FUNCTION_BLOCK FB_System_BHKW_921
VAR
	Pumpe_321: FB_PU;
	Stellventil_321: FB_SVs;
	Regelventil_321: FB_RV;
	BHKW_921: FB_BHKW;
	Zustandscheck: FB_System_BHKW_Zustandscheck;
	Logik: FB_System_BHKW_Logik;
	Ablaufsteuerung: FB_System_BHKW_Ablaufsteuerung;
	Timer1: TON;
	Timer_BHKW921_Pumpe321_Freigabe: TOF;
	Sollwertscheck: FB_System_BHKW_Sollwertscheck;
END_VAR
VAR_INPUT
	Freigabe_auto: BOOL := TRUE;
	Betrieb_Anford_auto: BOOL := FALSE;
	Regelung_Sollw_auto: REAL := 60;
END_VAR
VAR_OUTPUT
	{attribute 'OPC.UA.DA' := '1'}Steuerung: ST_System_BHKW_Steuerung; 
	{attribute 'OPC.UA.DA' := '1'}Stellwert: ST_System_BHKW_Stellwert; 
	{attribute 'OPC.UA.DA' := '1'}Zustand: ST_System_BHKW_Zustand; 		
	{attribute 'OPC.UA.DA' := '1'}Parameter: ST_System_BHKW_Parameter; 
END_VAR
VAR // added by the converter: edge detectors and wires of the graphical bodies
    _w1, _w2, _w3, _w4 : ANY;
END_VAR

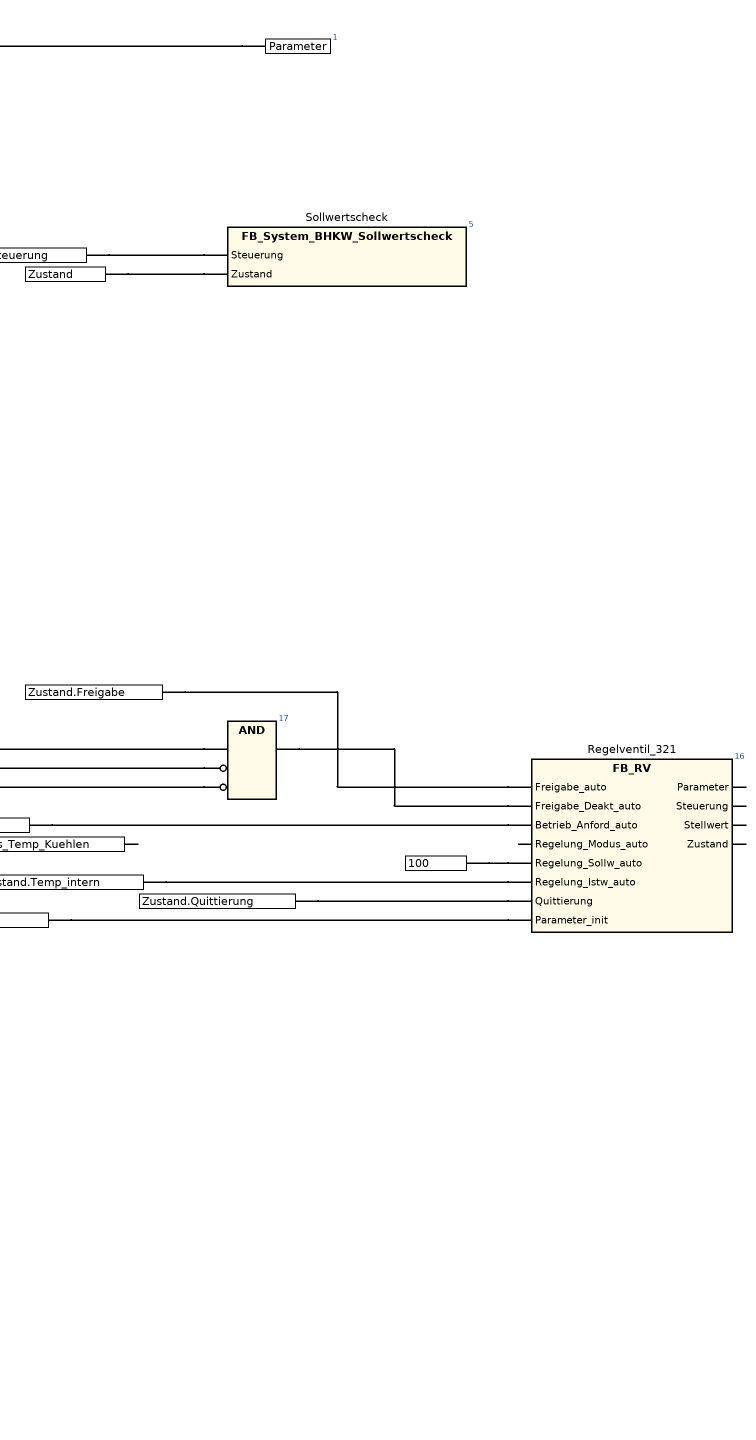
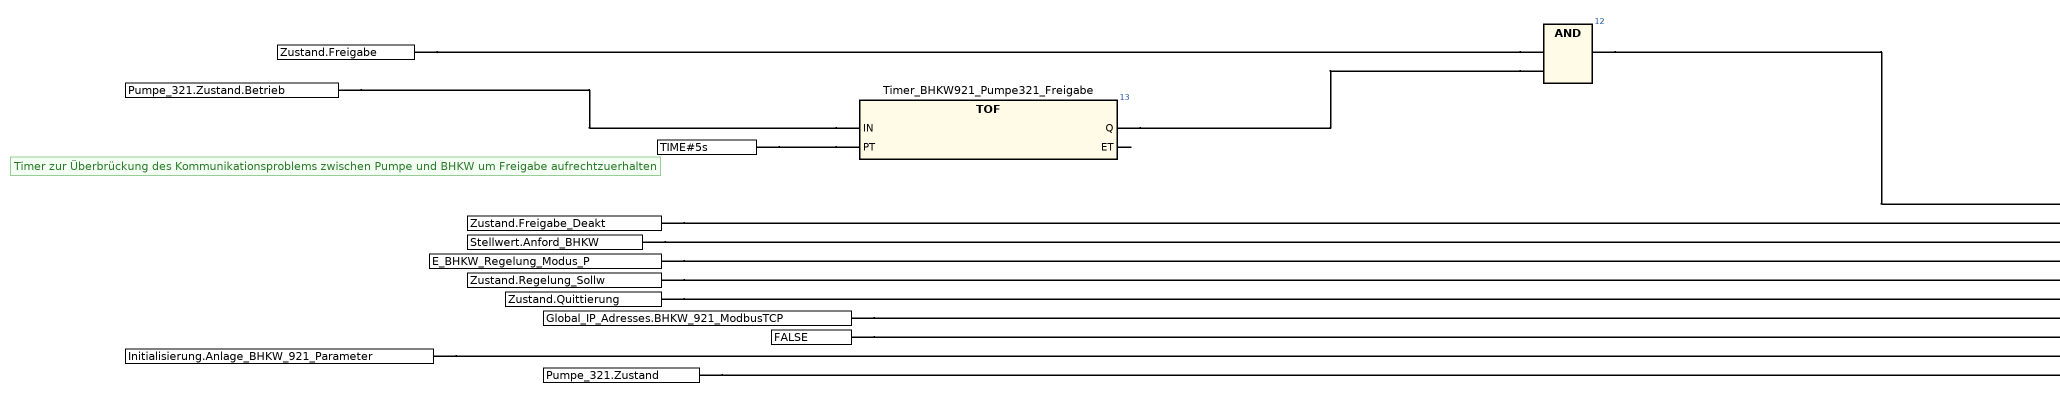
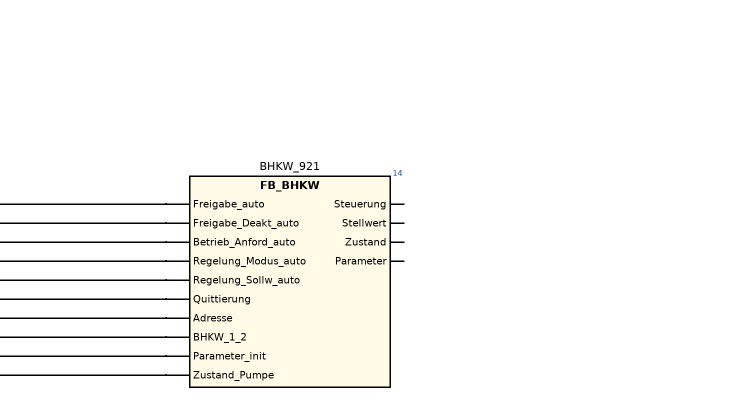
Steuerung.Freigabe.auto := Freigabe_auto;
Parameter := Initialisierung.System_BHKW_Parameter;
Steuerung.Freigabe_Deakt.auto := TRUE;
Steuerung.Betrieb_Anford.auto := Betrieb_Anford_auto;
Steuerung.Regelung_Sollw.auto := Regelung_Sollw_auto;
Sollwertscheck(Steuerung := Steuerung, Zustand := Zustand); // FB_System_BHKW_Sollwertscheck
Zustandscheck(
    Zustand_Stellventil := Stellventil_321.Zustand,
    Zustand_Pumpe := Pumpe_321.Zustand,
    Zustand_BHKW := BHKW_921.Zustand,
    Parameter_BHKW := BHKW_921.Parameter,
    Steuerung := Steuerung,
    Zustand := Zustand); // FB_System_BHKW_Zustandscheck
Logik(Parameter := Parameter, Steuerung := Steuerung, Zustand := Zustand); // FB_System_BHKW_Logik
Ablaufsteuerung(
    Zustand_Stellventil := Stellventil_321.Zustand,
    Zustand_Pumpe := Pumpe_321.Zustand,
    Zustand_BHKW := BHKW_921.Zustand,
    Zustand := Zustand,
    Stellwert := Stellwert,
    Steuerung := Steuerung,
    Parameter := Parameter); // FB_System_BHKW_Ablaufsteuerung
Pumpe_321(
    Freigabe_auto := Zustand.Freigabe,
    Freigabe_Deakt_auto := Zustand.Freigabe_Deakt AND NOT BHKW_921.Zustand.Betrieb,
    Betrieb_Anford_auto := Stellwert.Anford_Pumpe,
    Regelung_Modus_auto := SEL(TRUE, E_PU_Regelung_Modus_T_int, E_PU_Regelung_Modus_P),
    Regelung_Sollw_auto := _w1,
    Quittierung := Zustand.Quittierung,
    Parameter_init := Initialisierung.Pumpe_321_Parameter); // FB_PU
_w2 := Zustand.Freigabe AND Timer_BHKW921_Pumpe321_Freigabe.Q;
// Timer zur Überbrückung des Kommunikationsproblems zwischen Pumpe und BHKW um Freigabe aufrechtzuerhalten
Timer_BHKW921_Pumpe321_Freigabe(IN := Pumpe_321.Zustand.Betrieb, PT := TIME#5s); // TOF
BHKW_921(
    Freigabe_auto := _w2,
    Freigabe_Deakt_auto := Zustand.Freigabe_Deakt,
    Betrieb_Anford_auto := Stellwert.Anford_BHKW,
    Regelung_Modus_auto := E_BHKW_Regelung_Modus_P,
    Regelung_Sollw_auto := Zustand.Regelung_Sollw,
    Quittierung := Zustand.Quittierung,
    Adresse := Global_IP_Adresses.BHKW_921_ModbusTCP,
    BHKW_1_2 := FALSE,
    Parameter_init := Initialisierung.Anlage_BHKW_921_Parameter,
    Zustand_Pumpe := Pumpe_321.Zustand); // FB_BHKW
_w1 := SEL(TRUE, 40, 100);
Regelventil_321(
    Freigabe_auto := Zustand.Freigabe,
    Freigabe_Deakt_auto := _w3,
    Betrieb_Anford_auto := Stellwert.Anford_Stellventil,
    Regelung_Sollw_auto := 100,
    Regelung_Istw_auto := Pumpe_321.Zustand.Temp_intern,
    Quittierung := Zustand.Quittierung,
    Parameter_init := Initialisierung.Regelventil_321_Parameter); // FB_RV
_w3 := Zustand.Freigabe_Deakt AND NOT Pumpe_321.Zustand.Betrieb AND NOT BHKW_921.Zustand.Betrieb;
Stellventil_321(
    Freigabe_auto := Zustand.Freigabe,
    Freigabe_Deakt_auto := _w4,
    Stellung_Anford_auto := Stellwert.Anford_Stellventil,
    Quittierung := Zustand.Quittierung,
    Parameter_init := Initialisierung.Stellventil_321_Parameter); // FB_SVs
_w4 := Zustand.Freigabe_Deakt AND NOT Pumpe_321.Zustand.Betrieb AND NOT BHKW_921.Zustand.Betrieb;
// Zustand.Status_BHKW_ueberhitzt: input not connected
// E_RV_Regelung_Modus_Temp_Kuehlen: input not connected

END_FUNCTION_BLOCK

(* stored: Version 1.1.0.1, ProductVersion 3.1.4024.9
   POU FB_System_BHKW_921: Id {33e24615-b7cc-414f-82d9-9b8091608e05}, SpecialFunc None *)
